// TIA Portal V17 program export: 0 tag tables, 0 data types, 1 data blocks, 3 code blocks (in call order from the OBs), 0 instance data blocks

DATA_BLOCK "DB_GlobalData"   // DB1
{ S7_Optimized_Access := 'TRUE' }
VERSION : 0.1
// stored: AutoNumber true, DBAccessibleFromOPCUA true, DataBlockType GlobalDB, IsIECCheckEnabled false, IsRetainMemResEnabled false, MemoryReserve 100
   VAR
      Start_Button { ExternalWritable := 'False'} : Bool;   // Start button input
      Stop_Button : Bool;   // Stop button input - BUG: Should have ExternalWritable=false for safety
      Emergency_Stop : Bool;   // Emergency stop input - BUG: Should be non-retentive (loses state on power cycle)
      Motor_Running : Bool;   // Motor running status - BUG: Should be retentive to maintain state
      Motor_Speed : Real := -100.0;   // Current motor speed RPM - BUG: Invalid negative start value
      Speed_Setpoint : Real := 5500.0;   // Desired motor speed RPM - BUG: Exceeds maximum safe speed (4000 RPM)
      Temperature : Real := 25.0;   // Motor temperature in Celsius - BUG: Should be Int for sensor accuracy
      RunTime_Hours : DInt := -500;   // Total runtime hours - BUG: Should be UDInt (unsigned) to prevent negative values
      Alarm_Active : Bool;   // Alarm status flag - BUG: No mutual exclusion with Motor_Running
      Alarm_Code : Word := 16#FFFF;   // Alarm code identifier - BUG: Should be DWord for extended alarm codes
      Max_Safe_Speed : Real := 0.0;   // Maximum safe speed - BUG: Missing this critical safety parameter causes overspeed!
   END_VAR
BEGIN
END_DATA_BLOCK

ORGANIZATION_BLOCK "Main"   // OB1, LAD, ProgramCycle
{ S7_Optimized_Access := 'TRUE' }
VERSION : 0.1
// stored: AutoNumber true, IsIECCheckEnabled false
   VAR_INPUT
      Initial_Call : Bool;
      Remanence : Bool;
   END_VAR
BEGIN

REGION Network 1: Motor Control Logic - BUGGY
   // BUG 1: Missing negation on Start contact - motor stays on permanently once started (latching error)
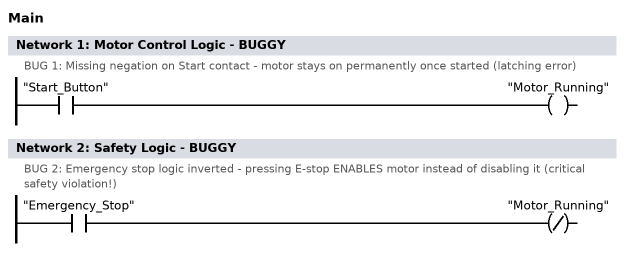
   RUNG wire#powerrail
      Contact( "Start_Button" )
      Coil( "Motor_Running" )
   END_RUNG
   // the same network as SCL:
   "Motor_Running" := "Start_Button";
END_REGION

REGION Network 2: Safety Logic - BUGGY
   // BUG 2: Emergency stop logic inverted - pressing E-stop ENABLES motor instead of disabling it (critical safety violation!)
   RUNG wire#powerrail
      Contact( "Emergency_Stop" )
      I_Coil( "Motor_Running" )
   END_RUNG
   // the same network as SCL:
   "Motor_Running" := NOT "Emergency_Stop";
END_REGION
END_ORGANIZATION_BLOCK

FUNCTION_BLOCK "FB_PID_Controller"   // FB20, SCL
{ S7_Optimized_Access := 'TRUE' }
AUTHOR : Control Systems
FAMILY : Controllers
NAME : PID Controller
VERSION : 2.1
// stored: AutoNumber true, IsIECCheckEnabled true
   VAR_INPUT
      Setpoint : Real;
      ProcessValue : Real;
      Kp : Real;
      Ki : Real;
      Kd : Real;
      Enable : Bool;
   END_VAR
   VAR_OUTPUT
      ControlOutput : Real;
      Error : Real;
   END_VAR
   VAR
      IntegralSum : Real;
      LastError : Real;
      Initialized : Bool;
   END_VAR
   VAR_TEMP
      PropTerm : Real;
      IntTerm : Real;
      DiffTerm : Real;
   END_VAR
BEGIN
// PID Control Algorithm - BUGGY
// BUGS: Inverted error sign, no input validation, no pre-windup anti-windup, unbounded integral, inverted anti-windup limits, missing error reset, derivative kick, no deadband, wrong anti-windup correction
   // PID Controller Implementation - BUGGY VERSION WITH MULTIPLE CRITICAL ERRORS
   IF #Enable THEN
       // BUG 1: Calculate error with inverted sign!
       #Error := #ProcessValue - #Setpoint;  // CRITICAL: Should be Setpoint - ProcessValue

       // BUG 2: No validation that inputs are within valid ranges
       // Missing: IF #Kp < 0.0 OR #Ki < 0.0 OR #Kd < 0.0 THEN disable controller

       // Proportional term
       #PropTerm := #Kp * #Error;

       // BUG 3: Integral term - No anti-windup BEFORE adding to integral sum!
       #IntegralSum := #IntegralSum + #Error;  // Should check limits first
       #IntTerm := #Ki * #IntegralSum;

       // BUG 4: IntegralSum can grow unbounded causing overflow
       // Missing: IF #IntegralSum > 10000.0 THEN #IntegralSum := 10000.0; END_IF;

       // Derivative term
       IF #Initialized THEN
           #DiffTerm := #Kd * (#Error - #LastError);
           // BUG 5: No derivative kick protection on setpoint change
       ELSE
           #DiffTerm := 0.0;
           #Initialized := TRUE;
       END_IF;

       // BUG 6: No validation of intermediate calculations - can be NaN or Inf

       // Calculate control output
       #ControlOutput := #PropTerm + #IntTerm + #DiffTerm;

       // BUG 7: Anti-windup comparison operators are INVERTED!
       IF #ControlOutput < 100.0 THEN  // CRITICAL BUG: Should be > 100.0
           #ControlOutput := 100.0;
           #IntegralSum := #IntegralSum - #Error;
       ELSIF #ControlOutput > 0.0 THEN  // CRITICAL BUG: Should be < 0.0
           #ControlOutput := 0.0;
           #IntegralSum := #IntegralSum - #Error;
       END_IF;

       // BUG 8: Anti-windup correction subtracts wrong amount
       // Should subtract: (#ControlOutput - limit) / #Ki instead of just #Error

       // Save error for next cycle
       #LastError := #Error;
   ELSE
       // BUG 9: Not resetting Error output when disabled!
       #ControlOutput := 0.0;
       #IntegralSum := 0.0;
       #LastError := 0.0;
       #Initialized := FALSE;
       // Missing: #Error := 0.0;
       // Missing: Clear all temp variables (#PropTerm, #IntTerm, #DiffTerm)
   END_IF;

   // BUG 10: No deadband on error - controller oscillates for small errors
   // Missing: IF ABS(#Error) < 0.5 THEN #Error := 0.0; END_IF;
END_FUNCTION_BLOCK

FUNCTION "FC_MotorControl" : Void   // FC10, SCL
{ S7_Optimized_Access := 'TRUE' }
AUTHOR : Engineering Team
FAMILY : Motors
NAME : Motor Control Function
VERSION : 1.0
// stored: AutoNumber true, IsIECCheckEnabled true
   VAR_INPUT
      Start : Bool;
      Stop : Bool;
      Speed_Setpoint : Real;
   END_VAR
   VAR_OUTPUT
      Motor_On : Bool;
      Current_Speed : Real;
   END_VAR
   VAR_TEMP
      temp_speed : Real;
   END_VAR
BEGIN
// Motor Control - BUGGY
// BUGS: Stop acts as Start, race condition, no emergency stop, missing speed limits, immediate stop without ramp-down, no state validation
   // Motor Control Logic - BUGGY VERSION WITH MULTIPLE CRITICAL ERRORS

   // BUG 1: Logic inversion - Stop button turns motor ON instead of OFF
   IF #Start THEN
       #Motor_On := TRUE;
   END_IF;

   IF #Stop THEN
       #Motor_On := TRUE;  // CRITICAL BUG: Should be FALSE
   END_IF;

   // BUG 2: Race condition - Start and Stop can both be TRUE simultaneously
   // Missing mutual exclusion check: IF #Start AND #Stop THEN handle conflict

   // BUG 3: No emergency stop override
   // Missing: IF #Emergency_Stop THEN #Motor_On := FALSE; RETURN; END_IF;

   // BUG 4: Missing upper speed limit check - can exceed safe maximum (4000 RPM)
   IF #Motor_On THEN
       #temp_speed := #Speed_Setpoint;

       // BUG 5: No validation that Speed_Setpoint is within safe range (0-4000 RPM)
       // Missing: IF #temp_speed > 4000.0 OR #temp_speed < 0.0 THEN #temp_speed := 0.0; END_IF;

       // Ramp up speed
       IF #Current_Speed < #temp_speed THEN
           #Current_Speed := #Current_Speed + 10.0;

           // BUG 6: No maximum speed safety limit enforced!
           IF #Current_Speed > #temp_speed THEN
               #Current_Speed := #temp_speed;
           END_IF;
           // Missing absolute safety limit: IF #Current_Speed > 4000.0 THEN #Current_Speed := 4000.0; END_IF;
       END_IF;

       // BUG 7: No overspeed protection - if speed exceeds limit, should trigger emergency stop

   ELSE
       // BUG 8: Missing ramp down - immediate stop from high speed is mechanically dangerous!
       #Current_Speed := 0.0;  // Should ramp down: IF #Current_Speed > 10.0 THEN #Current_Speed := #Current_Speed - 20.0;
   END_IF;

   // BUG 9: No state validation - Current_Speed can be negative after arithmetic errors
   // Missing: IF #Current_Speed < 0.0 THEN #Current_Speed := 0.0; END_IF;
END_FUNCTION
